(* PLC project Untitled1, Beckhoff Automation GmbH TwinCAT PLC Control 3.5.13.20 *)
(* stored: creationDateTime 2022-07-20T15:22:55.2280327, modificationDateTime 2022-07-20T15:22:55.2280327 *)

{attribute 'qualified_only'}
{attribute 'strict'}
TYPE eFirmerVendorEvent1 : (eNoInfo := 0, ePowerCurtailmentFromExternalCommand := 1, ePowerLimitationFromFrequencyWatt := 2, ePowerLimitationFromHighAverageGridVoltage := 3, ePowerLimitationFromAntiIslandingProtection := 4, ePowerLimitationFromGridCurrentRatingLimitation := 5, ePowerLimitationForHighTemperature := 6, ePowerLimitationForHighDCVoltage := 7, ePowerLimitationFromRampRateConnectionRamp := 9, ePowerLimitationFromMomentaryCessation := 10, ePowerLimitationFromRampRateNormalRampUp := 11, ePowerLimitationFromVoltWatt := 12, ePowerLimitationFromCapabilityRating := 13);
END_TYPE
